hm	14. mar. 2009	rev 1.2
	removed double assignments

*)

END_FUNCTION_BLOCK

// POUs/Logic/gate logic/SHR1
FUNCTION SHR1 : DWORD
VAR_INPUT
	IN : DWORD;
	N : INT;
END_VAR
VAR CONSTANT
	temp : DWORD := 16#FFFF_FFFF;
END_VAR

(*
version 1.1	27 dec 2007
programmer 	hugo
tested by		tobias

SHR1 shifts N bits to the right filling the new bits with 1

*)

SHR1 := SHL(temp,32-N) OR SHR(IN,N);

(* revision history
hm	14.9.2007		rev 1.0
	original version

hm	27. dec 2007	rev 1.1
	changed code for better performance

*)

END_FUNCTION

// POUs/Mathematical/SIGMOID
FUNCTION SIGMOID : REAL
VAR_INPUT
	X : REAL;
END_VAR


(*
version 1.2	10. mar. 2009
programmer 	hugo
tested by		tobias

this function calculates the sigmoid function

*)

IF X > 20.0 THEN
	SIGMOID := 1.0;
ELSIF x < -85.0 THEN
	SIGMOID := 0.0;
ELSE
	SIGMOID := 1.0 / (1.0 + EXP(-X));
END_IF;


(* revision history
hm	10.12.2007		rev 1.0
	original version

hm	11. mar. 2008		rev 1.1
	extended range of valid inputs to +inv / -inv

hm 10. mar. 2009		rev 1.2
	real constants updated to new systax using dot																																																																																																																																																																																																																																																																																																																																																																																																																																																																																																																																																																																																																																																																																																																																																																																																																																																																																																																																																																																																																																																											

*)

END_FUNCTION

// POUs/Mathematical/SIGN_I
FUNCTION SIGN_I : BOOL
VAR_INPUT
	IN : DINT;
END_VAR


(*
version 1.3	27. oct. 2008
programmer 	hugo
tested by	tobias

this function return true if the integer input is negative

*)

SIGN_I := in.31;

(* revision history
hm 3.3.2007	rev 1.1
	changed method of function for better compatibility to other systems

hm	1.12.2007	rev 1.2
	changed code to improve performance

hm	27. oct. 2008	rev 1.3
	changed type of input to dint

*)

END_FUNCTION

// POUs/Engineering/automation/SIGNAL_4
FUNCTION_BLOCK SIGNAL_4
VAR_INPUT
	IN1 : BOOL;
	IN2 : BOOL;
	IN3 : BOOL;
	IN4 : BOOL;
	TS : TIME;
END_VAR
VAR_INPUT CONSTANT
	S1 : BYTE := 2#1111_1111;
	S2 : BYTE := 2#1111_0000;
	S3 : BYTE := 2#1010_1010;
	S4 : BYTE := 2#1010_0000;
END_VAR
VAR_OUTPUT
	Q : BOOL;
END_VAR
VAR
	sig : SIGNAL;
END_VAR

(*
version 1.0	13 dec 2007
programmer 	hugo
tested by		tobias

this function generates one out of 4 signals specified by bit patterns S1 .. S4.
the selected pattern will be shifted with the step time TS.
In1 has higher priority then In2 which has higher priority then IN3 and in4 has the lowest priority.
ts defaults to 128 ms if not specified.
*)

(* an alarm is present read system time first *)
(* check if an alarm is present if yes set sig to the alarm pattern otherwise exit the routine *)
IF in1 THEN
	sig(in := TRUE, sig := s1, TS := TS);
ELSIF in2 THEN
	sig(in := TRUE, sig := s2, TS := TS);
ELSIF in3 THEN
	sig(in := TRUE, sig := s3, TS := TS);
ELSIF in4 THEN
	sig(in := TRUE, sig := s4, TS := TS);
ELSE
	sig(in := FALSE);
END_IF;

(* set the output *)
Q := sig.Q;


(* revision history
hm	13.12.2007		rev 1.0
	original version

*)

END_FUNCTION_BLOCK

// POUs/Mathematical/SINC
FUNCTION SINC : REAL
VAR_INPUT
	X : REAL;
END_VAR


(*
version 1.2	10. mar. 2009
programmer 	hugo
tested by		tobias

this function calculates the sinc function.

*)

IF X = 0.0 THEN
	SINC := 1.0;
ELSE
	SINC := SIN(x) / x;
END_IF;


(* revision histroy
hm	11. mar. 2008	rev 1.0
	original version

hm	1.12.2007	rev 1.1
	changed code to improove performance

hm 10. mar. 2009	rev 1.2
	real constants updated to new systax using dot																																																																																																																																																																																																																																																																																																																																																																																																																																																																																																																																																																																																																																																																																																																																																																																																																																																																																																																																																																																																																																																											

*)

END_FUNCTION

// POUs/Mathematical/Geometry/SPHERE_V
FUNCTION SPHERE_V : REAL
VAR_INPUT
	rx : REAL;
END_VAR


(*
version 1.2	22. feb 2008
programmer 	hugo
tested by		tobias

sphere_V calculates the Volume of a Sphere


*)

sphere_V := 4.188790205 * Rx * RX * RX;

(* revision histroy
hm	16. oct 2007	rev 1.0
	original version

hm	4. dec 2007		rev 1.1
	changed code for better performance

hm	22. feb 2008		rev 1.2
	changed code for better performance
*)

END_FUNCTION

// POUs/Engineering/automation/SRAMP
FUNCTION_BLOCK SRAMP
VAR_INPUT
	X : REAL;
	A_UP : REAL;
	A_DN :REAL;
	VU_MAX : REAL;
	VD_MAX : REAL;
	LIMIT_HIGH : REAL;
	LIMIT_LOW : REAL;
	RST : BOOL;
END_VAR
VAR_OUTPUT
	Y : REAL;
	V : REAL;
END_VAR
VAR
	cycle_time : TC_S;
	init: BOOL;
END_VAR


(*
	version 1.1	11. mar. 2009
	programmer 	hugo
	tested by		tobias

RAMPS generates output signal which are slew rate and acceleration controlled.

*)

(* read the system_time in microseconds *)
cycle_time();

(* assure range of inputs *)
A_up := MAX(0.0, A_UP);
A_dn := MIN(0.0, A_dn);
VU_max := MAX(0.0, VU_max);
VD_max := MIN(0.0, VD_MAX);

(* calculate the output offset *)
IF rst OR NOT init THEN
	init := TRUE;
	Y := 0.0;
	V := 0.0;
ELSIF X = Y THEN
	v := 0.0;
ELSIF X > Y THEN
	(* output is too low >> ramp up and brake at the end *)
	(* accelerate the speed and limit to vu_max *)
	v := MIN(v + A_UP * cycle_time.TC, vu_max);
	(* calculate the max speed to be able to brake and select the lowest *)
	v := MIN(SQRT((Y-X) * 2.0 * A_DN), v);
	(* calculate the output and obey limits *)
	y := LIMIT(limit_low, y + MIN(v * cycle_time.TC, X-Y), limit_high);
ELSIF X < Y THEN
	(* output is too high >> ramp dn and brake at the end *)
	(* accelerate the speed and limit to vd_max *)
	v := MAX(v + A_DN * cycle_time.TC, vd_max);
	(* calculate the max speed to be able to brake and select the lowest *)
	v := MAX(-SQRT((Y-X) * 2.0 * A_UP), v);
	(* calculate the output and obey limits *)
	y := LIMIT(limit_low, y + MAX(v * cycle_time.TC, X-Y), limit_high);
END_IF;


(* revision history
hm	13. mar. 2008	rev 1.0
	original version

hm	11. mar. 2009	rev 1.1
	real constants updated to new systax using dot																																																																																																																																																																																																																																																																																																																																																																																																																																																																																																																																																																																																																																																																																																																																																																																																																																																																																																																																																																																																																																																											

*)

END_FUNCTION_BLOCK

// POUs/Engineering/measurements/TC_S
FUNCTION_BLOCK TC_S

VAR_OUTPUT
	TC : REAL;
END_VAR
VAR
	init: BOOL;
	tx: DWORD;
	last: DWORD;
END_VAR

(*
	version 1.2	11. mar. 2009
	programmer 	hugo
	tested by		tobias

TC_S delivers the time it was last called on the output TC in seconds.

*)

(* read system timer *)
tx := T_PLC_US();

IF NOT init THEN
	init := TRUE;
	TC := 0.0;
ELSE
	tc := DWORD_TO_REAL(tx - last)*1.0E-6;
END_IF;
last := tx;

(* revision history
hm	13. mar. 2008	rev 1.0
	original version

hm	16. mar 2008	rev 1.1
	added type conversion to avoid warnings under codesys 3.0

hm	11. mar. 2009	rev 1.2
	changed real constants to use dot syntax

*)

END_FUNCTION_BLOCK

// POUs/Logic/memory/STACK_16
FUNCTION_BLOCK STACK_16
VAR_INPUT
	Din : DWORD;
	E : BOOL := TRUE;
	RD : BOOL;
	WD : BOOL;
	RST : BOOL;
END_VAR
VAR_OUTPUT
	Dout : DWORD;
	EMPTY : BOOL := TRUE;
	FULL : BOOL;
END_VAR
VAR
	stack : ARRAY[0..n] OF DWORD;
	pt : INT;
END_VAR
VAR CONSTANT
	n : INT := 15;	(* changing this value will chage the number of stored elements in the fifo *)
END_VAR


(*
version 2.0	25. jul 2009
programmer 	hugo
tested by		oscat

16 Dword STACK memory

*)

IF RST THEN
	(* asynchronous reset for the fifo *)
	pt := 0;
	EMPTY := TRUE;
	FULL := FALSE;
	Dout := 0;
ELSIF E THEN
	IF NOT EMPTY AND RD THEN
		(* read one element *)
		pt := pt - 1;
		Dout := stack[pt];
		EMPTY := pt = 0;
		FULL := FALSE;
	END_IF;
	IF NOT FULL AND WD THEN
		(* write one element *)
		stack[pt] := Din;
		pt := pt + 1;
		FULL := pt > n;
		EMPTY := FALSE;
	END_IF;
END_IF;


(* revision history
hm	4. aug. 2006	rev 1.0
	original version

hm	19. feb 2008	rev 1.1
	performance improvements

hm	17. oct. 2008	rev 1.2
	deleted unnecessary init with 0

hm	27. oct. 2008	rev 1.3
	optimized performance

hm	25. jul 2009	rev 2.0
	changed inputs to allow simultsaneous read and write
*)

END_FUNCTION_BLOCK

// POUs/Logic/memory/STACK_32
FUNCTION_BLOCK STACK_32
VAR_INPUT
	Din : DWORD;
	E : BOOL := TRUE;
	RD : BOOL;
	WD : BOOL;
	RST : BOOL;
END_VAR
VAR_OUTPUT
	Dout : DWORD;
	EMPTY : BOOL := TRUE;
	FULL : BOOL;
END_VAR
VAR
	stack : ARRAY[0..n] OF DWORD;
	pt : INT;
END_VAR
VAR CONSTANT
	n : INT := 31;	(* changing this value will chage the number of stored elements in the fifo *)
END_VAR


(*
version 2.0	25. jul 2009
programmer 	hugo
tested by		oscat

32 Dword STACK memory
*)

IF RST THEN
	(* asynchronous reset for the fifo *)
	pt := 0;
	EMPTY := TRUE;
	FULL := FALSE;
	Dout := 0;
ELSIF E THEN
	IF NOT EMPTY AND RD THEN
		(* read one element *)
		pt := pt - 1;
		Dout := stack[pt];
		EMPTY := pt = 0;
		FULL := FALSE;
	END_IF;
	IF NOT FULL AND WD THEN
		(* write one element *)
		stack[pt] := Din;
		pt := pt + 1;
		FULL := pt > n;
		EMPTY := FALSE;
	END_IF;
END_IF;


(* revision history
hm	4. aug. 2006	rev 1.0
	original version

hm	19. feb 2008	rev 1.1
	performance improvements

hm	17. oct. 2008	rev 1.2
	deleted unnecessary init with 0

ks	27. oct. 2008	rev 1.3
	optimized performance

hm	25. jul 2009	rev 2.0
	changed inputs to allow simultsaneous read and write

*)

END_FUNCTION_BLOCK

// POUs/Engineering/signal processing/STAIR
FUNCTION STAIR : REAL
VAR_INPUT
	X : REAL;
	D : REAL;
END_VAR


(*
version 1.4	10. mar. 2009
programmer 	oscat
tested by		tobias

the function stair converts an anlog input signal to a staircase like output.
D is the step width for the output signal.
if D = 0 then the output follows the input without a chage.
*)

IF D > 0.0 THEN
	STAIR := DINT_TO_REAL(REAL_TO_DINT(X / D)) * D;
ELSE
	STAIR := X;
END_IF;



(* revision history
hm	28 jan 2007		rev 1.0
	original version

hm	27 dec 2007		rev 1.1
	changed code for better performance

hm	6. jan 2008		rev 1.2
	further performance improvement

hm	26. oct. 2008		rev 1.3
	optimized code

hm	10. mar. 2009	rev 1.4
	real constants updated to new systax using dot

*)

END_FUNCTION

// POUs/Engineering/signal processing/STAIR2
FUNCTION_BLOCK STAIR2
VAR_INPUT
	X : REAL;
	D : REAL;
END_VAR
VAR_OUTPUT
	Y: REAL;
END_VAR


(*
version 1.4	10. mar. 2009
programmer 	hugo
tested by		oscat

the function stair2 converts an anlog input signal to a staircase like output.
D is the step width for the output signal. the output will use D as a hysteresis for a stairchange.
if D = 0 then the output follows the input without a chage.
*)

IF D > 0.0 THEN
	IF X >= Y + D OR X <= Y - D THEN Y := FLOOR(X/D) * D; END_IF;
ELSE
	Y := X;
END_IF;



(* revision history
hm	28 jan 2007		rev 1.0
	original version

hm	27. dec 2007	rev 1.1
	changed code for better performance

hm	30. jun. 2008	rev 1.2
	added type conversions to avoid warnings under codesys 3.0																																																																																																																																																																																																																																																											

ks	26. oct. 2008	rev 1.3
	improved code

hm	10. mar. 2009	rev 1.4
	real constants updated to new systax using dot

*)

END_FUNCTION_BLOCK

// POUs/Logic/FF pulse triggered/STORE_8
FUNCTION_BLOCK STORE_8
VAR_INPUT
	Set : BOOL;
	D0,D1, D2, D3, D4, D5, D6, D7 : BOOL;
	Clr : BOOL;
	Rst : BOOL;
END_VAR
VAR_OUTPUT
	Q0, Q1, Q2, Q3, Q4, Q5, Q6, Q7 : BOOL;
END_VAR
VAR
	edge: BOOL;
END_VAR

(*
version 1.2	14. mar. 2009
programmer 	hugo
tested by		oscat

Store_4 stores up to 4 boolean inputs until a reset is clearing the outputs.
the respective output is set with a true at the respective input and stays true until a reset is generated.
a set input is used to set all outputs true at the same time, independent of their inputs.
a clear input is used to reset only the lowest priority of the outputs one at a time.
the lowest priority is q3.

*)

IF rst OR set THEN
	q0 := NOT rst;
	q1 := q0;
	q2 := q0;
	q3 := q0;
	q4 := q0;
	q5 := q0;
	q6 := q0;
	q7 := q0;
ELSE
	IF D0 THEN Q0 := TRUE; END_IF;
	IF D1 THEN Q1 := TRUE; END_IF;
	IF D2 THEN Q2 := TRUE; END_IF;
	IF D3 THEN Q3 := TRUE; END_IF;
	IF D4 THEN Q4 := TRUE; END_IF;
	IF D5 THEN Q5 := TRUE; END_IF;
	IF D6 THEN Q6 := TRUE; END_IF;
	IF D7 THEN Q7 := TRUE; END_IF;

	IF clr AND NOT edge THEN
		IF q0 THEN q0 := FALSE;
		ELSIF q1 THEN q1 := FALSE;
		ELSIF q2 THEN q2 := FALSE;
		ELSIF q3 THEN q3 := FALSE;
		ELSIF q4 THEN q4 := FALSE;
		ELSIF q5 THEN q5 := FALSE;
		ELSIF q6 THEN q6 := FALSE;
		ELSE q7 := FALSE;
		END_IF;
	END_IF;
	edge := clr;
END_IF;


(* revision history
hm	25.12.2007	rev 1.0
	original version

hm	30. oct. 2008	rev 1.1
	optimized performance

hm	14. mar. 2009	rev 1.2
	removed double assignments

*)

END_FUNCTION_BLOCK

// POUs/Logic/gate logic/SWAP_BYTE
FUNCTION SWAP_BYTE : WORD
VAR_INPUT
	IN : WORD;
END_VAR


(*
version 1.0	4 feb 2008
programmer 	hugo
tested by		tobias

This function swaps the high and low byte of the word in.

*)

SWAP_BYTE := ROL(in,8);


(* revision history
hm		4. feb 2008	rev 1.0
	original version

*)

END_FUNCTION

// POUs/Logic/gate logic/SWAP_BYTE2
FUNCTION SWAP_BYTE2 : DWORD
VAR_INPUT
	IN : DWORD;
END_VAR


(*
version 1.0	4 feb 2008
programmer 	hugo
tested by		tobias

This function reverses the byte order in the dword.

*)

Swap_Byte2 := (ROR(in,8) AND 16#FF00FF00) OR (ROL(in,8) AND 16#00FF00FF);

(* revision history
hm		4. feb 2008	rev 1.0
	original version

*)

END_FUNCTION

// POUs/Building/electrical/SWITCH_I
FUNCTION_BLOCK SWITCH_I
VAR_INPUT
	set : BOOL;
	in : BOOL;
	rst : BOOL;
END_VAR
VAR_INPUT CONSTANT
	T_debounce : TIME := T#10ms;
	T_reconfig : TIME := T#1s;
	T_on_max : TIME := T#0h;
END_VAR
VAR_OUTPUT
	Q : BOOL;
END_VAR
VAR
	state : BYTE;
	edge : BOOL;
	r_edge : BOOL;
	T_on : TIME;
	tx: TIME;
END_VAR

(*
version 1.1	15 sep 2007
programmer 	oscat
tested by	oscat

this is an intelligent switch interface which has an autodetect feature for in and it will detect the type of switch connected automatically
the input can be connected to low active pulses, high active pulses and on/off switch.
it will automatically adjust to the correct type without manual adjustment
a configurable debounce timer will debounce input signals
if t_on_max is set to anything other then 0 the output will be turned off after the max on time is reached.

*)

(* read system time *)
tx := DWORD_TO_TIME(T_PLC_MS());

(* asynchronous set and reset first *)
IF set AND NOT rst THEN
	Q := TRUE;
	T_on := tx;
ELSIF rst THEN
	Q := FALSE;
(* check FOR input edge AND start debounce timer *)
ELSIF (in XOR edge) AND NOT (state = 1) THEN
	state := 1;
	T_on := Tx;
(* edge was detected and debounce time elapsed *)
ELSIF (state = 1) AND (Tx - t_debounce >= T_on) THEN
	state := 2;
	(* react on rising or falling edge depending on r_edge *)
	IF r_edge XOR in THEN Q := NOT Q; END_IF;
(* wait for T_reconfig and adjust r_edge *)
ELSIF state = 2 AND Tx - t_reconfig >= T_on THEN
	r_edge := in;
END_IF;
IF Q AND T_on_max > t#0ms AND Tx >= T_on + T_on_max THEN
	Q := FALSE;
END_IF;
edge := in;

(* revision history

hm	4 aug 2006	rev 1.0
	original version

hm	15.9.2007	rev 1.1
	replaced Time() with T_PLC_MS for compatibility and performance reasons

*)

END_FUNCTION_BLOCK

// POUs/Building/electrical/SWITCH_X
FUNCTION_BLOCK SWITCH_X
VAR_INPUT
	IN1 : BOOL;
	IN2 : BOOL;
	IN3 : BOOL;
	IN4 : BOOL;
	IN5 : BOOL;
	IN6 : BOOL;
END_VAR
VAR_OUTPUT
	Q1 : BOOL;
	Q2 : BOOL;
	Q3 : BOOL;
	Q4 : BOOL;
	Q5 : BOOL;
	Q6 : BOOL;
	Q31 : BOOL;
	Q41 : BOOL;
	Q51 : BOOL;
	Q61 : BOOL;
	Q32 : BOOL;
	Q42 : BOOL;
	Q52 : BOOL;
	Q62 : BOOL;
END_VAR
VAR_INPUT CONSTANT
	t_debounce : TIME := t#50ms;
END_VAR
VAR
	init : BOOL;
	T1, T2, T3, T4, T5, T6 : TOF;
	tx: TIME;
	x1: BOOL;
	x2: BOOL;
	E1, E2 : BOOL;
END_VAR

(*
version 1.0	15 Feb 2007
programmer 	oscat
tested by	oscat

*)

(* initialize on startup *)
IF NOT init THEN
	init := TRUE;
	IF t_debounce < t#50ms THEN tx := t#50ms; ELSE tx := t_debounce; END_IF;
	T1(PT := Tx);
	T2(PT := Tx);
	T3(PT := Tx);
	T4(PT := Tx);
	T5(PT := Tx);
	T6(PT := Tx);
ELSE
	Q1 := FALSE;
	Q2 := FALSE;
	Q3 := FALSE;
	Q4 := FALSE;
	Q5 := FALSE;
	Q6 := FALSE;
	Q31 := FALSE;
	Q41 := FALSE;
	Q51 := FALSE;
	Q61 := FALSE;
	Q32 := FALSE;
	Q42 := FALSE;
	Q52 := FALSE;
	Q62 := FALSE;
END_IF;

(* read inputs and debounce *)
	T1(IN := IN1);
	T2(IN := IN2);
	T3(IN := IN3);
	T4(IN := IN4);
	T5(IN := IN5);
	T6(IN := IN6);

(* detect edge of IN1 and IN2 *)
IF t1.Q AND NOT E1 THEN X1 := TRUE; END_IF;
IF t2.Q AND NOT E2 THEN X2 := TRUE; END_IF;

IF t1.Q THEN
	IF t3.q THEN
		q31 := TRUE;
		X1 := FALSE;
	ELSIF t4.q THEN
		q41 := TRUE;
		X1 := FALSE;
	ELSIF t5.q THEN
		q51 := TRUE;
		X1 := FALSE;
	ELSIF t6.q THEN
		q61 := TRUE;
		X1 := FALSE;
	END_IF;
ELSIF t2.Q THEN
	IF t3.q THEN
		q32 := TRUE;
		X2 := FALSE;
	ELSIF t4.q THEN
		q42 := TRUE;
		X2 := FALSE;
	ELSIF t5.q THEN
		q52 := TRUE;
		X2 := FALSE;
	ELSIF t6.q THEN
		q62 := TRUE;
		X2 := FALSE;
	END_IF;
(* in1 was active alone *)
ELSIF NOT T1.Q AND E1 AND X1 THEN
	Q1 := TRUE;
	X1 := FALSE;
ELSIF NOT T2.Q AND E2 AND X2 THEN
	Q2 := TRUE;
	X2 := FALSE;
ELSIF T3.Q THEN
	Q3 := TRUE;
ELSIF T4.Q THEN
	Q4 := TRUE;
ELSIF T5.Q THEN
	Q5 := TRUE;
ELSIF T6.Q THEN
	Q6 := TRUE;
END_IF;

(* save state of in1 and in2 *)
E1 := T1.Q;
E2 := T2.Q;

END_FUNCTION_BLOCK

// POUs/Building/HLK/T_AVG24
FUNCTION_BLOCK T_AVG24
VAR_INPUT
	TS : INT;
	DTI : DT;
	RST : BOOL;
END_VAR
VAR_INPUT CONSTANT
	T_FILTER : TIME := T#10m;
	SCALE : REAL := 1.0;
	OFS : REAL;
END_VAR
VAR_OUTPUT
	TA : REAL;
	TP : BOOL;
END_VAR
VAR_IN_OUT
	T24 : REAL;
	T24_MAX : REAL;
	T24_MIN : REAL;
END_VAR
VAR
	samples : ARRAY[0..47] OF INT;
	pos : INT;
	init: BOOL;
	ft1 : FILTER_I;
	sum : DINT;
	last: DT;
END_VAR
VAR
	tmp_max : INT;
	tmp_min : INT;
	i: INT;
END_VAR

(*
version 1.2	13. mar. 2009
programmer 	hugo
tested by		oscat

this function calculates the averaged daytime temperature by taking 48 samples over one day.
a trigger tp will be true for one cycle when the output is updated.
using the input scale the outputs can be adjusted to different scales.

*)

(* first filter the sensor readings *)
ft1(X := TS, T := T_FILTER);

IF rst OR NOT init THEN
	init := TRUE;
	IF T24 = -1000.0 THEN t24 := INT_TO_REAL(ft1.Y) * 0.1; END_IF;
	FOR pos := 0 TO 47 DO
		samples[pos] := REAL_TO_INT(T24 * 10.0);
	END_FOR;
	pos := 0;
	sum := INT_TO_DINT(samples[0]) * 48;
	(* calculate the output value *)
	TA := (INT_TO_REAL(ft1.Y) * 0.1 + OFS) * SCALE;
	T24 := (DINT_TO_REAL(sum) * 0.00208333333333 + OFS) * SCALE;
	tp := TRUE;
ELSIF DT_TO_DWORD(dti) / 60 MOD 30 = 0 AND DTI > last THEN
	(* make sure we onlyexecute once every 30 mins *)
	last := DTI + T#1m;
	(* sample the temperature every 30 mins and store in ring buffer samples *)
	(* sum always holds the sum of the array *)
	(* subtract the oldest sample from sum *)
	sum := sum - INT_TO_DINT(samples[pos]);
	(* strore the new sample *)
	samples[pos] := ft1.Y;
	(* add the new sample to sum *)
	sum := sum + INT_TO_DINT(samples[pos]);
	(* increment the counter for the next sample *)
	pos := INC1(pos, 48);
	(* calculate the output value *)
	TA := (INT_TO_REAL(ft1.Y) * 0.1 + OFS) * SCALE;
	T24 := (DINT_TO_REAL(sum) * 0.00208333333333 + OFS) * SCALE;
	(* calculate the min and max over the last 24 hours *)
	tmp_max := -32000;
	tmp_min := 32000;
	FOR i := 0 TO 47 DO
		tmp_max := MAX(tmp_max, samples[i]);
		tmp_min := MIN(tmp_min, samples[i]);
	END_FOR;
	T24_MAX := (INT_TO_REAL(tmp_max) * 0.1 + OFS) * SCALE;
	T24_MIN := (INT_TO_REAL(tmp_min) * 0.1 + OFS) * SCALE;
	tp := TRUE;
ELSE
	tp := FALSE;
END_IF;





(* revision history
hm	3. nov. 2008	rev 1.0
	original version

hm	8. feb. 2009	rev 1.1
	changes sign of OFS
	added outputs t24_min and t24_max

hm	13. mar. 2009	rev 1.2
	improved code
*)

END_FUNCTION_BLOCK

// POUs/Mathematical/TANC
FUNCTION TANC : REAL
VAR_INPUT
	X : REAL;
END_VAR


(*
version 1.1	10. mar. 2009
programmer 	hugo
tested by		oscat

this function calculates the tanc function.

*)

IF X = 0.0 THEN
	TANC := 1.0;
ELSE
	TANC := TAN(x) / x;
END_IF;


(* revision histroy
hm	23. oct. 2008	rev 1.0
	original version

hm 10. mar. 2009	rev 1.1
	real constants updated to new systax using dot																																																																																																																																																																																																																																																																																																																																																																																																																																																																																																																																																																																																																																																																																																																																																																																																																																																																																																																																																																																																																																																											

*)

END_FUNCTION

// POUs/Mathematical/TANH
FUNCTION TANH : REAL
VAR_INPUT
	X : REAL;
END_VAR


(*
version 1.3	10. mar. 2009
programmer 	hugo
tested by		tobias

this function calculates the tangens hyperbolicus

*)

IF X > 20.0 THEN
	TANH := 1.0;
ELSIF X < -20.0 THEN
	TANH := -1.0;
ELSE
	TANH := 1.0 - 2.0 / (EXP(2.0 * x) + 1.0);
END_IF;


(* revision hisdtory
hm		12.1.2007		rev 1.0
	original version

hm		1.12.2007		rev 1.1
	changed code to improve performance

hm		10. mar 2008	rev 1.2
	corrected an error in formula
	extended range of valid inputs to +/- INV

hm 10. mar. 2009	rev 1.3
	real constants updated to new systax using dot																																																																																																																																																																																																																																																																																																																																																																																																																																																																																																																																																																																																																																																																																																																																																																																																																																																																																																																																																																																																																																																											

*)

END_FUNCTION

// POUs/Engineering/automation/TANK_LEVEL
FUNCTION_BLOCK TANK_LEVEL
VAR_INPUT
	LEVEL : BOOL;
	LEAK : BOOL;
	ACLR : BOOL;
END_VAR
VAR_INPUT CONSTANT
	MAX_VALVE_TIME : TIME;
	LEVEL_DELAY_TIME : TIME;
END_VAR
VAR_OUTPUT
	VALVE : BOOL;
	ALARM : BOOL;
	STATUS : BYTE;
END_VAR
VAR
	cx : ACTUATOR_COIL;
	tn : TON;
	tl : TONOF;
	open: BOOL;
END_VAR


(*
version 1.1	24 jul 2009
programmer 	hugo
tested by		tobias

*)

(* preprocess the level information *)
tl(in := level, T_ON := level_delay_time, T_OFF := level_delay_time);
open := tl.Q;

(* start logic *)
IF ALARM THEN
	(* check for ACLR if ALARM is present *)
	IF ACLR THEN
		ALARM := FALSE;
		STATUS := 101; (* aclr pressed *)
		cx(in := FALSE);
	END_IF;
	RETURN;
ELSIF LEAK THEN
	(* leakeage detected *)
	cx(in := FALSE);
	ALARM := TRUE;
	STATUS := 1;	(* leakeage error *)
ELSIF open THEN
	(* valve needs to be opened because level is too low *)
	cx(in := TRUE);
	STATUS := 102; (* valve open by low level *)
ELSE
	(* valve needs to be closed *)
	cx(in := FALSE);
	STATUS := 100; (* valve idle *)
END_IF;

(* check if valve is open too long and generate alarm if necessary *)
tn(in := cx.out AND (MAX_VALVE_TIME > T#0s), PT := MAX_VALVE_TIME);
IF tn.Q THEN
	ALARM := TRUE;
	STATUS := 2; (* overtime error *)
	cx(in := FALSE);
END_IF;

(* set output signal *)
VALVE := cx.out;


(* revision history
hm 27. feb 2007	rev 1.0
	original version

hm	24. jul 2009	rev 1.1
	changed parameters of tonof

*)

END_FUNCTION_BLOCK

// POUs/Logic/generators/TONOF
FUNCTION_BLOCK TONOF
VAR_INPUT
	IN : BOOL;
	  T_ON,T_OFF : TIME;
END_VAR
VAR_OUTPUT
	Q : BOOL;
END_VAR
VAR
   X : TON;
   old: BOOL;
   mode: BOOL;
END_VAR

(*
version 1.2	21. jul 2009
programmer 	hugo
tested by		tobias

TONOF generated a TON and TOF Delay for the Input N TON (T1) and TOF (T2) can be configured separately
*)

IF IN XOR old THEN
  X(IN := FALSE, PT := SEL(IN,T_OFF,T_ON));
  mode := IN;
  old := IN;
END_IF;
X(IN := TRUE);
IF X.Q THEN Q := mode;END_IF;

(* revision history
hm	10. dec 2007	rev 1.0
	original version

hm	17. sep. 2007	rev 1.1
	improved performance

hm	21. jul. 2009	rev 1.2
	fixed a timing probelm


*)

END_FUNCTION_BLOCK

// POUs/Building/HLK/TANK_VOL1
FUNCTION TANK_VOL1 : REAL
VAR_INPUT
	TR : REAL;
	TL : REAL;
	H : REAL;
END_VAR


(*
version 1.0	10. Mar 2010
programmer 	hugo
tested by		tobias

TANK_VOL1 calculates the volume of a tubular tank filled to level H.


*)

TANK_VOL1 := CIRCLE_SEG(TR, H) * TL;


(* revision histroy
hm	10. mar 2010	rev 1.0
	original version

*)

END_FUNCTION

// POUs/Building/HLK/TANK_VOL2
FUNCTION TANK_VOL2 : REAL
VAR_INPUT
	TR : REAL;
	H : REAL;
END_VAR


(*
version 1.0	10. Mar 2010
programmer 	hugo
tested by		tobias

TANK_VOL2 calculates the volume of a spherical tank filled to level H.

*)

TANK_VOL2 := math.PI * H * H * (TR - H/3.0);

(* revision histroy
hm	10. mar 2010	rev 1.0
	original version

*)

END_FUNCTION

// POUs/Engineering/measurements/TC_MS
FUNCTION_BLOCK TC_MS

VAR_OUTPUT
	TC : DWORD;
END_VAR
VAR
	init: BOOL;
	tx: DWORD;
	last: DWORD;
END_VAR

(*
	version 1.0	13 mar 2008
	programmer 	hugo
	tested by		tobias

TC_MS delivers the time it was last called on the output TC in Milliseconds.

*)

(* read system timer *)
tx := T_PLC_MS();

IF NOT init THEN
	init := TRUE;
	TC := 0;
ELSE
	tc := tx - last;
END_IF;
last := tx;

(* revision history
hm		13. mar. 2008	rev 1.0
	original version

*)

END_FUNCTION_BLOCK

// POUs/Engineering/measurements/TC_US
FUNCTION_BLOCK TC_US

VAR_OUTPUT
	TC : DWORD;
END_VAR
VAR
	init: BOOL;
	tx: DWORD;
	last: DWORD;
END_VAR

(*
	version 1.0	13 mar 2008
	programmer 	hugo
	tested by		tobias

TC_US delivers the time it was last called on the output TC in Microseconds.

*)

(* read system timer *)
tx := T_PLC_US();

IF NOT init THEN
	init := TRUE;
	TC := 0;
ELSE
	tc := tx - last;
END_IF;
last := tx;

(* revision history
hm		13. mar. 2008	rev 1.0
	original version

*)

END_FUNCTION_BLOCK

// POUs/Building/HLK/TEMP_EXT
FUNCTION_BLOCK TEMP_EXT
VAR_INPUT
	t_ext1 : REAL;
	t_ext2 : REAL;
	t_ext3 : REAL;
	t_ext_config : BYTE;
	dt_in : DT;
END_VAR
VAR_INPUT CONSTANT
	t_ext_min : REAL := -40.0;
	t_ext_max : REAL := 60.0;
	t_ext_default : REAL := -10.0;
	heat_period_start : DATE := D#1970-9-1;
	heat_period_stop : DATE := D#1970-4-30;
	cool_period_start : DATE := D#1970-4-1;
	cool_period_stop : DATE := D#1970-9-30;
	heat_start_temp_day : REAL := 15.0;
	heat_start_temp_night : REAL := 10.0;
	heat_stop_temp : REAL := 18.0;
	cool_start_temp_day : REAL := 26.0;
	cool_start_temp_night : REAL := 26.0;
	cool_stop_temp : REAL := 24.0;
	start_day : TOD := tod#09:00;
	start_night : TOD := tod#21:00;
	CYCLE_TIME : TIME := t#10m;
END_VAR
VAR_OUTPUT
	t_ext : REAL;
	heat : BOOL;
	cool : BOOL;
END_VAR
VAR
	tx: TIME;
	last_run: TIME;
	init: BOOL;
	cool_start: DATE;
	cool_stop: DATE;
	heat_start: DATE;
	heat_stop: DATE;
	xdate: DATE;
	day: BOOL;
END_VAR


(*
version 1.3	13. mar. 2009
programmer 	hugo
tested by		oscat

temp_ext measures and processes ext temperature and decides if heating or cooling is needed.

 the measurement of t_ext has 3 inputs which can be configured in different ways:
	t_ext_config = 0 means the ext temp is the avg of the 3 external temperatures, this mode is the default mode.
	t_ext_config = 1 means t_ext1 is used.
	t_ext_config = 2 means t_ext1 is used.
	t_ext_config = 3 means t_ext1 is used.
	t_ext_config = 4 means t_ext_default is used.
	t_ext_config = 5 means the lowest of the 3 external temperatures is used.
	t_ext_config = 6 means the higest externnal temperature is used.
	t_ext_config = 7 means the midlle external temperature is used, if there are only two working, the lowest is used.
	in any config mode, an external temperature higher then t_ext_max or lower then t_ext_min is ignored to prevent from temperatures caused by broken sensors or wires.
	if no external temperature is available, a default value (t_ext_default) is used.
	if you have only one external sensor, connect the 3 inputs to the same sensor, or select the right input with t_ext_config.

heating or cooling is enabled during heating / cooling period when the day or night start temperature is reached for at least the specified delay time and will be disabled after the stop temperature is reached. 
t_ext output can be used by other modules to determine the correct system temperature for heating or cooling.

*)

IF NOT init THEN
	init := TRUE;
	heat_start := SET_DATE(1972,MONTH_OF_DATE(heat_period_start),DAY_OF_MONTH(heat_period_start));
	heat_stop := SET_DATE(1972,MONTH_OF_DATE(heat_period_stop),DAY_OF_MONTH(heat_period_stop));
	cool_start := SET_DATE(1972,MONTH_OF_DATE(cool_period_start),DAY_OF_MONTH(cool_period_start));
	cool_stop := SET_DATE(1972,MONTH_OF_DATE(cool_period_stop),DAY_OF_MONTH(cool_period_stop));
END_IF;

(* read system time *)
tx := DWORD_TO_TIME(T_PLC_MS());

(* for efficiency exit isf this program has been executed less then 1min ago *)
IF tx - last_run < cycle_time THEN RETURN; END_IF;

(* calculate frequently used variables *)
xdate := SET_DATE(1972,MONTH_OF_DATE(DT_TO_DATE(dt_in)),DAY_OF_MONTH(DT_TO_DATE(dt_in)));
day := DT_TO_TOD(dt_in) >= start_day AND  DT_TO_TOD(dt_in) < start_night;

(* read the correct external temperature depending on the t_ext_config setting *)
t_ext := MULTI_IN(t_ext1, t_ext2, t_ext3, t_ext_default, t_ext_min, t_ext_max, t_ext_config);

(* dtermine heating *)
IF (heat_start <= heat_stop AND xdate >= heat_start AND xdate <= heat_stop) OR (heat_start > heat_stop AND (xdate >= heat_start OR xdate <= heat_stop)) THEN
	(* heating period id true check for temperature *)
	IF day AND t_ext <= heat_start_temp_day THEN
		heat := TRUE;
	ELSIF NOT day AND t_ext <= heat_start_temp_night THEN
		heat := TRUE;
	ELSIF t_ext >= heat_stop_temp THEN
		heat := FALSE;
	END_IF;
ELSE
	heat := FALSE;
END_IF;

(* dtermine cooling *)
IF (cool_start <= cool_stop AND xdate >= cool_start AND xdate <= cool_stop) OR (cool_start > cool_stop AND (xdate >= cool_start OR xdate <= cool_stop)) THEN
	(* cooling period is true check for temperature *)
	IF day AND t_ext >= cool_start_temp_day THEN
		cool := TRUE;
	ELSIF NOT day AND t_ext >= cool_start_temp_night THEN
		cool := TRUE;
	ELSIF t_ext <= cool_stop_temp THEN
		cool := FALSE;
	END_IF;
ELSE
	cool := FALSE;
END_IF;

last_run := tx;

(* revision history
hm	6 dec 2006	rev 1.0
	original version

hm	15.9.2007		rev 1.1
	replaced Time() with T_PLC_MS for compatibility and performance reasons

hm	7. oct. 2008	rev 1.2
	changed name of function month to month_of_date

hm	13. mar. 2009	rev 1.3
	real constants updated to new systax using dot

*)

END_FUNCTION_BLOCK

// POUs/Engineering/sensor/TEMP_NI
FUNCTION TEMP_NI : REAL
VAR_INPUT
	Res : REAL;
	R0 : REAL;
END_VAR


(*
version 1.5	10. mar. 2009
programmer 	hugo
tested by		tobias

this function returns the temperature for a nickel sensor in a range from -60..+180 °C *)

TEMP_NI := (SQRT(0.30085225 - 2.66E-3 * (R0 - Res)) - 0.5485) * 751.8796992;


(* revision history

hm 24.1.2007		rev 1.1
	deleted unused variable A, B, C

hm 10.9.2007		rev 1.2
	changed accuracy to 0.02 degrees to improove performace

hm 17. 12 2007	rev 1.3
	improovements for better performance and higher accuracy

hm	6. jan 2008	rev 1.4
	further performance improvement

hm	10. mar. 2009	rev 1.5
	removed nested comments

*)

END_FUNCTION

// POUs/Engineering/sensor/TEMP_NTC
FUNCTION TEMP_NTC : REAL
VAR_INPUT
	RES : REAL;
	RN : REAL;
	B : REAL;
END_VAR


(*
version 1.1	11. mar. 2009
programmer 	hugo
tested by		tobias

this function returs the temperature for a NTC sensor for a range from 0..85 °C.
RN is the resistance at 25 °C and B is a constant for the given sensor.

*)

IF res > 0.0 THEN
	TEMP_NTC := B * 298.15 / (B + LN(RES / RN) * 298.15) -273.15;
END_IF;


(* revision history

hm 30. dec. 2008	rev 1.0
	original version

hm	11. mar. 2009	rev 1.1
	changed real constants to use dot syntax

*)

END_FUNCTION

// POUs/Engineering/sensor/TEMP_PT
FUNCTION TEMP_PT : REAL
VAR_INPUT
	Res : REAL;
	R0 : REAL;
END_VAR
VAR CONSTANT
	A : REAL := 3.9083E-3 ;
	B : REAL := -5.775E-7;
	accuracy : REAL := 0.01;
END_VAR
VAR
	step: REAL := 50.0;
	X: REAL;
	Y: REAL;
	t1: REAL;
	pt : POINTER TO DWORD;
END_VAR

(*
version 1.7	11. mar. 2009
programmer 	hugo
tested by		oscat

this function returs the temperature for a platinum sensor for a range from -200..+850 °C *)

X := A * R0;
Y := B * R0;
IF Res >= R0 THEN
	t1 := X * X - 4.0 * Y * (R0 - Res);
	IF t1 < 0.0 THEN
		TEMP_PT := 10000.0;
	ELSE
		TEMP_PT := (-X + SQRT(t1)) / (2.0 * Y);
	END_IF;
ELSE
	pt := ADR(step);
	(* since the formula cannot be solved this is a successive approximation *)
	TEMP_PT := -100.0;
	WHILE step > accuracy DO
		(* test if result greater or less *)
		IF RES_PT(TEMP_PT, R0) < res THEN TEMP_PT := TEMP_PT + step; ELSE TEMP_PT := TEMP_PT - step; END_IF;
		pt^ := pt^ - 8388608;  (* this is a super fast divide by 2 method for non floating point CPUs *)
		(* the alternative code: step := step * 0.5; *)
	END_WHILE;
END_IF;

(* revision history

rev 1.1 hm 24.1.2007	
	deleted unused variable C

rev 1.2 hm 10.9.2007
	reduced accuracy to 0.02 to shorten execution time

rev 1.3	hm	2. dec 2007
	changed code for better performance

rev	1.4	hm	23. dec 2007
	avoid a negative square root if input values are wrong

rev 1.5 hm	5. jan 2008
	replaced / 2 with * 0.5 for better performance

hm	31. oct. 2008	rev 1.6
	improved performance

hm	11. mar. 2009	rev 1.7
	changed real constants to use dot syntax

*)

END_FUNCTION

// POUs/Engineering/sensor/TEMP_SI
FUNCTION TEMP_SI : REAL
VAR_INPUT
	Res : REAL;
	RS : REAL;
	TS : REAL;
END_VAR


(*
version 1.5	10. mar. 2009
programmer 	hugo
tested by		tobias

this function returs the temperature for a silicon sensor for a range from -60..+180 °C
for example KTY10 RS at TS normally 25 °C
*)

TEMP_SI := (-7.64E-3 + SQRT(Res / RS * 6.64E-5 - 0.803E-5)) * 30120.48193 + TS;



(* revision history

hm 24.1.2007		rev 1.1
	the function would only work for TS = 25, now it works for other values of ts.

hm 10.9.2007		rev 1.2
	changed the function to use successive approcimation to avoid an error generated by a sqrt from a negative result.
	changed accuracy to 0.02 degrees to shorten execution time

hm 17. 12 2007	rev 1.3
	improovements for better performance

hm	6. jan 2008	rev 1.4
	further performance improvement

hm	10. mar. 2009	rev 1.5
	removed nested comments

*)

END_FUNCTION

// POUs/String/TICKER
FUNCTION_BLOCK TICKER

VAR_INPUT
	N : INT;
	PT : TIME;
END_VAR

VAR_IN_OUT
	Text : STRING(STRING_LENGTH);
END_VAR

VAR_OUTPUT
	Display : STRING(STRING_LENGTH);
END_VAR
VAR
	delay : TP;
	step : INT;
END_VAR

(*
version 1.2	29. mar. 2008
programmer 	hugo
tested by		tobias

Ticker sends a substring of text with length N every TD Milliseconds to generate a ticker. 

*)


(* generate next ticker when delay is low *)
IF N < LEN(text) THEN
	IF NOT delay.Q THEN
		(* increase step for next tick *)
		step := step + 1;
		IF step > LEN(text) THEN step := 1; END_IF;
		(* extract dispay from text *)
		display := MID(text, N, step);
		(* set delay timer for next tick *)
		delay(in := TRUE, PT := PT);
	ELSE;
		(* execute delay timer *)
		delay(in := FALSE);
	END_IF;
ELSE
	display := text;
END_IF;
(* revision history
hm	4. dec. 2007	rev 1.0
	original version

hm	15. dec. 2007	rev 1.1
	step now starts at 1 instaed of 0

hm	29. mar. 2008	rev 1.2
	changed STRING to STRING(STRING_LENGTH)
*)

END_FUNCTION_BLOCK

// POUs/Building/electrical/TIMER_2
FUNCTION_BLOCK TIMER_2
VAR_INPUT
	DT_in : DT;
	start : TOD;
	duration : TIME;
	mode : BYTE;
	HOLIDAY : BOOL;
END_VAR
VAR_OUTPUT
	Q : BOOL;
END_VAR
VAR
	last_check : TIME;
	dat : DATE;
	daytime : TOD;
	activation: TIME;
	tx: TIME;
	enabled: BOOL;
	init: BOOL;
	wday : INT;
END_VAR

VAR RETAIN
	run_date : DATE;
END_VAR

(*
version 1.4	20. oct. 2008
programmer 	oscat
tested by	oscat

this timer generated programmabe output pulses per day, week, month and so on.
the mode input determines on which days the timer will be active.
	mode = 0			never
	mode = 1..7			monday .. sunday
	mode = 11			every day
	mode = 12			every second day
	mode = 13			every 3rd day
	mode = 14			every 4th day
	mode = 15			every 5th day
	mode = 16 			every 6th day
	mode = 20			only monday - friday
	mode = 21			only sat - sunday
	mode = 22			workdays only
	mode = 23			holidays and weekend
	mode = 24			holidays only
	mode = 25			every 1st day of the month
	mode = 26			every last day of the month
	mode = 27			every 31 of december
	mode = 28			every 1st of january

a holiday input can be used to supply holiday information to the module.
*)

(* read system time *)
tx := DWORD_TO_TIME(T_PLC_MS());

IF NOT init THEN
	init := TRUE;
	last_check := tx - t#100ms;
END_IF;

(* for performance resons exit if execution is not necessary *)
IF tx - last_check < T#100ms THEN RETURN; END_IF;

(* calculate temp variables *)
dat := DT_TO_DATE(dt_in);
daytime := DT_TO_TOD(dt_in);
wday := DAY_OF_WEEK(dat);

(* calculate if any action is necessary today *)
CASE mode OF
	1..7:	(* mondays to fridays *)
		enabled := wday = BYTE_TO_INT(mode);
	11:	(* every day *)
		enabled := TRUE;
	12..16:	(* every nth day *)
		enabled := (DATE_TO_DWORD(dat)/86400) MOD (mode - 10) = 0;
	20:	(* monday - friday *)
		enabled := wday <= 5;
	21:	(* saturday and sunday *)
		enabled := wday > 5;
	22: (* workdays only *)
		enabled := wday <= 5 AND NOT holiday;
	23:	(* holidays and weekends *)
		enabled := wday > 5 OR holiday;
	24:	(* holidays only *)
		enabled := holiday;
	25:	(* 1st day of the month *)
		enabled := DAY_OF_MONTH(dat) = 1;
	26:	(* last day of month *)
		enabled := DAY_OF_MONTH(dat + t#1d) = 1;
	27:	(* 31st of december *)
		enabled := DAY_OF_MONTH(dat) = 31 AND MONTH_OF_DATE(dat) = 12;
	28:	(* 1st of january *)
		enabled := DAY_OF_YEAR(dat) = 1;
ELSE
	enabled := FALSE;
END_CASE;

(* set output if necessary *)
IF enabled AND NOT Q AND daytime >= start AND run_date <> dat THEN
	Q := TRUE;
	activation := tx;
	run_date := dat;
ELSIF Q AND tx - activation >= duration THEN
	Q := FALSE;
END_IF;
last_check := Tx;


(* revision history
hm 22.2.2007		rev 1.1
	changed VAR RETAIN PERSISTENT to VAR RETAIN for better compatibility
	wago lon contollers do not support persisitent

hm	15.9.2007		rev 1.2
	replaced Time() with T_PLC_MS for compatibility and performance reasons

hm	7. oct. 2008	rev 1.3
	changed function month to month_of_date

hm	20. oct. 2008	rev 1.4
	improved performance
	deleted unnecessary trunc

hm	22. dec. 2008	rev 1.5
	make sure timer_2 is executed in the first cycle

*)

END_FUNCTION_BLOCK

// POUs/Building/electrical/TIMER_EVENT_DECODE
FUNCTION TIMER_EVENT_DECODE : TIMER_EVENT
VAR_INPUT
	EVENT : STRING(STRING_LENGTH);
	LANG :	INT;
END_VAR
VAR
	pos: INT;
	start : INT;
	stop: INT;
	pt : POINTER TO ARRAY[1..255] OF BYTE;
	step: INT;
	tmp : STRING(60);
END_VAR



(*
version 1.1	25. oct. 2008
programmer 	hugo
tested by	oscat

STRING_TO_TIMER_EVENT converts a string to a timer event structure.

*)

(* a timer event is specified as follows:
	$typ;ch;day;start;duration;land;lor#
$ 		= start of definition
typ 	= type of definition	(number)
channel	= channel number		(number)
day 	= day number			(number)
start	= start time			(time of day)
duration= duration of event		(time)
land	= mask for output AND	(8bit value)
lor		= mask for ourput OR	(8bit value)
#		= end of definition
*)

(* check for start and ending character *)
IF (LEFT(event,1) <> '<') AND (RIGHT(event,1) <> '>') THEN RETURN; END_IF;
stop := LEN(event);
pt := ADR(event);
start := 2;

(* parse the string for next ; *)
FOR pos := 2 TO stop DO
	IF pt^[pos] = 59 OR pt^[pos] = 62 THEN
		tmp := MID(event, pos - start, start);
		CASE step OF
			0:	(* read type *)
				TIMER_EVENT_DECODE.typ := FSTRING_TO_BYTE(tmp);

			1:	(* read channel *)
				TIMER_EVENT_DECODE.channel := FSTRING_TO_BYTE(tmp);

			2:	(* read day *)
				IF IS_CC(tmp,'0123456789abcdefABCDEF#') THEN
					TIMER_EVENT_DECODE.day := FSTRING_TO_BYTE(tmp);
				ELSIF TIMER_EVENT_DECODE.typ = 2 THEN
					TIMER_EVENT_DECODE.DAY := FSTRING_TO_WEEK(tmp, LANG);
				ELSE
					TIMER_EVENT_DECODE.DAY := INT_TO_BYTE(FSTRING_TO_WEEKDAY(tmp, LANG));
				END_IF;

			3:	(* read start *)
				TIMER_EVENT_DECODE.start := STRING_TO_TOD(tmp);

			4:	(* read duaration *)
				TIMER_EVENT_DECODE.duration := STRING_TO_TIME(tmp);

			5:	(* read land *)
				TIMER_EVENT_DECODE.land := FSTRING_TO_BYTE(tmp);

			6:	(* read lor *)
				TIMER_EVENT_DECODE.LOR := FSTRING_TO_BYTE(tmp);
		END_CASE;
		start := pos + 1;
		step := step + 1;
	END_IF;
END_FOR;




(* revision history
hm	17. jun 2008	rev 1.0
	original version

hm	25. oct. 2008	rev 1.1
	adding input lang for language selection
*)

END_FUNCTION

// POUs/Building/electrical/TIMER_EXT
FUNCTION_BLOCK TIMER_EXT
VAR_INPUT
	ENA : BOOL := TRUE;
	ON : BOOL;
	OFF : BOOL;
	MAN : BOOL;
	SWITCH : BOOL;
	DT_IN : DT;
	SUN_RISE : TOD;
	SUN_SET : TOD;
	HOLIDAY : BOOL;
END_VAR
VAR_INPUT CONSTANT
	T_DEBOUNCE : TIME := T#100ms;
	T_RISE_START : TIME;
	T_RISE_STOP : TIME;
	T_SET_START : TIME;
	T_SET_STOP : TIME;
	T_DAY_START : TOD;
	T_DAY_STOP : TOD;
	ENABLE_SATURDAY : BOOL;
	ENABLE_SUNDAY : BOOL;
	ENABLE_HOLIDAY : BOOL;
END_VAR
VAR_OUTPUT
	Q : BOOL;
	STATUS: BYTE;
END_VAR
VAR
	mx : MANUAL_2;
	deb : DEBOUNCE;
	tdx: TOD;
	wdx: INT;
	tc : TIME;
	tx: DWORD;
	tl: DWORD;
	qx: BOOL;
	init: BOOL;
END_VAR

(*
version 1.1	6. nov. 2008
programmer 	oscat
tested by	tobias

TIMER_EXT is a twilight timer.
the timer can be programmed to switch lights or other equippment or during twilight times.
in addition to the automatik mode the timer can be stopped and started by a switch at any given time.
An enable input ENA can be used for external control.
two inputs ON and OFF can be used to statically control the output.
the timer can be programmed to work on saturdays, sundays and holidays if required.

*)

(* lösche die millisekunden bei sunrise und sunset *)
SUN_RISE := DWORD_TO_TOD(TOD_TO_DWORD(SUN_RISE) / 1000 * 1000);
SUN_SET := DWORD_TO_TOD(TOD_TO_DWORD(SUN_SET) / 1000 * 1000);

(* measure cycle time tc and make sure this circuitry is not called more then once in 200ms*)
tx := T_PLC_MS();
IF NOT init THEN
	init := TRUE;
	tl := tx;
END_IF;
tc := DWORD_TO_TIME(tx - tl);
IF tc < t#200ms THEN RETURN; END_IF;
tl := tx;

(* debounce *)
deb(in := SWITCH, TD := T_DEBOUNCE, PM := TRUE);

(* read time of day and strip off all milliseconds *)
tdx := DT_TO_TOD(dt_in);
wdx := DAY_OF_WEEK(DT_TO_DATE(dt_in));

(* automatic output control *)
IF deb.Q THEN
	qx := NOT qx;
	status := 110;
ELSIF holiday AND NOT enable_holiday THEN
	qx := FALSE;
ELSIF wdx = 6 AND NOT enable_saturday THEN
	qx := FALSE;
ELSIF wdx = 7 AND NOT enable_sunday THEN
	qx := FALSE;
ELSIF T_day_start > TOD#00:00 AND tdx - T_DAY_START <= tc THEN
	(* turn on at specified daytime *)
	qx := TRUE;
	status := 111;
ELSIF T_DAY_STOP > TOD#00:00 AND tdx - T_DAY_STOP <= tc THEN
	(* turn off at specific daytime *)
	qx := FALSE;
	status := 112;
ELSIF T_RISE_START > T#0s AND tdx - SUN_RISE + T_RISE_START <= tc THEN
	(* turn on before sunrise *)
	qx := TRUE;
	status := 113;
ELSIF T_RISE_STOP > T#0s AND tdx - SUN_RISE - T_RISE_STOP <= tc THEN
	(* turn off after sunrise *)
	qx := FALSE;
	status := 114;
ELSIF T_SET_start > T#0s AND tdx - SUN_SET + T_SET_START <= tc THEN
	(* turn on before sunset *)
	qx := TRUE;
	status := 115;
ELSIF T_SET_STOP > t#0s AND tdx - SUN_SET - T_SET_STOP <= tc THEN
	(* turn off after sunset *)
	qx := FALSE;
	status := 116;
END_IF;


(* mnaual and output control *)
mx(in := qx, ena := ENA, on := ON, off := OFF, man := MAN);
Q := mx.Q;

(* set the status output *)
IF mx.STATUS > 100 THEN status := mx.STATUS; END_IF;



(*
hm 	7. oct. 2008	rev 1.0
	original version

hm	6. nov. 2008	rev 1.1
	added default = true for ena input
*)

END_FUNCTION_BLOCK

// POUs/Building/electrical/TIMER_P4
FUNCTION_BLOCK TIMER_P4
VAR_INPUT
	DTIME : DT;
	TREF_0 : TOD;
	TREF_1 : TOD;
	HOLY : BOOL;
	L0, L1, L2, L3 : BOOL;
	OFS : BYTE;
	ENQ : BOOL;
	MAN : BOOL;
	MI : BYTE;
	RST : BOOL;
END_VAR
VAR_IN_OUT
	PROG : ARRAY[0..array_max] OF TIMER_EVENT;
END_VAR
VAR_OUTPUT
	Q0, Q1, Q2, Q3 : BOOL;
	STATUS : BYTE;
END_VAR
VAR CONSTANT
	array_max : INT := 63;
	channel_max : INT := 3;
END_VAR
VAR
	day_start : DT;
	start : DT;
	event : TIMER_EVENT;
	pos : INT;
	last_execute: DT;
	current_day : DINT;
	mask: BYTE;
	ma : ARRAY[0..channel_max] OF BYTE;
	mo : ARRAY[0..channel_max] OF BYTE;
	qn : ARRAY[0..channel_max] OF BOOL;
	qs : ARRAY[0..channel_max] OF BOOL;
	channel: INT;
	tx: TOD;
END_VAR


(*
version 1.4	26. jan. 2011
programmer 	hugo
tested by	oscat

TIMER_P4 is a programmable universal timer.
*)

(* for performance reasons we only execute the code at the beginning of a new second *)

IF RST THEN
	(* reset all events to last active on 1.1.1970 *)
	last_execute := DT#1970-1-1-00:00;
	FOR pos := 0 TO ARRAY_MAX DO
		IF (PROG[pos].CHANNEL >= OFS) AND (PROG[pos].CHANNEL < (OFS + 4)) THEN PROG[pos].LAST := last_execute; END_IF;
	END_FOR;

	(* reset all set markers and logic masks *)
	FOR pos := 0 TO channel_max DO
		qs[pos] := FALSE;
	END_FOR;

(* normal operation *)
ELSIF dtime <> last_execute THEN
	(* save the actual second for next execution test *)
	last_execute := DTIME;

	(* calculate dt for the start of the day to be used in comparisons *)
	day_start := DATE_TO_DT(DT_TO_DATE(DTIME));

	(* set all qn to FALSE *)
	FOR pos := 0 TO channel_max DO qn[pos] := FALSE; END_FOR;

	(* search the array PROG for timer events *)
	FOR pos := 0 TO ARRAY_MAX DO
		event := prog[pos];
		channel := event.CHANNEL - OFS;
		IF (event.TYP > 0) AND (channel >= 0) AND (channel <= channel_max) THEN
			ma[channel] := event.LAND;
			mo[channel] := event.LOR;
			CASE event.TYP OF
				1:	(* daily event *)
					start := day_start + TOD_TO_TIME(event.start);
					qn[channel] := dtime >= start AND dtime <= start + event.DURATION;

				2: 	(* event by selected weekdays *)
					IF (SHR(BYTE#128, DAY_OF_WEEK(DT_TO_DATE(Dtime))) AND event.DAY) > 0 THEN
						start := day_start + TOD_TO_TIME(event.start);
						qn[channel] := dtime >= start AND dtime <= start + event.DURATION;
					END_IF;

				3:	(* event every N days *)
					IF current_day MOD event.DAY = 0 THEN
						start := day_start + TOD_TO_TIME(event.start);
						qn[channel] := dtime >= start AND dtime <= start + event.DURATION;
					END_IF;

				10:	(* weekly event exactly once a week the weekday is specified in day, 1= mo *)
					IF DAY_OF_WEEK(DT_TO_DATE(DTIME)) = BYTE_TO_INT(event.DAY) THEN
						start := day_start + TOD_TO_TIME(event.start);
						qn[channel] := dtime >= start AND dtime <= start + event.DURATION;
					END_IF;

				20:	(* monthly event *)
					IF DAY_OF_MONTH(DT_TO_DATE(DTIME)) = BYTE_TO_INT(event.DAY) THEN
						start := day_start + TOD_TO_TIME(event.start);
						qn[channel] := dtime >= start AND dtime <= start + event.DURATION;
					END_IF;

				21:	(* event on last day of month *)
					IF DT_TO_DATE(DTIME) = MONTH_END(DT_TO_DATE(dtime)) THEN
						start := day_start + TOD_TO_TIME(event.start);
						qn[channel] := dtime >= start AND dtime <= start + event.DURATION;
					END_IF;

				30:	(* yearly event on a specific day specified in day *)
					IF DAY_OF_YEAR(DT_TO_DATE(DTIME)) = BYTE_TO_INT(event.DAY) THEN
						start := day_start + TOD_TO_TIME(event.start);
						qn[channel] := dtime >= start AND dtime <= start + event.DURATION;
					END_IF;

				31:	(* event on last day of year *)
					IF DT_TO_DATE(DTIME) = YEAR_END(YEAR_OF_DATE(DT_TO_DATE(dtime))) THEN
						start := day_start + TOD_TO_TIME(event.start);
						qn[channel] := dtime >= start AND dtime <= start + event.DURATION;
					END_IF;

				40:	(* event on leap days *)
					IF LEAP_DAY(DT_TO_DATE(dtime)) THEN
						start := day_start + TOD_TO_TIME(event.start);
						qn[channel] := dtime >= start AND dtime <= start + event.DURATION;
					END_IF;

				41: (* event on holidays *)
					IF HOLY THEN
						start := day_start + TOD_TO_TIME(event.start);
						qn[channel] := dtime >= start AND dtime <= start + event.DURATION;
					END_IF;

				42: (* event on holidays and weekends *)
					IF (Holy OR (DAY_OF_WEEK(DT_TO_DATE(dtime)) = 6) OR (DAY_OF_WEEK(DT_TO_DATE(dtime)) = 7)) THEN
						start := day_start + TOD_TO_TIME(event.start);
						qn[channel] := dtime >= start AND dtime <= start + event.DURATION;
					END_IF;

				43:	(* event on workdays Mo-FR and no holiday *)
					IF DAY_OF_WEEK(DT_TO_DATE(dtime)) < 6 THEN
						start := day_start + TOD_TO_TIME(event.start);
						qn[channel] := dtime >= start AND dtime <= start + event.DURATION;
					END_IF;

				50: (* event after reference time *)
					CASE prog[pos].DAY OF
						0:	tx := tref_0;
						1:	tx := tref_1;
					ELSE
						tx := TOD#00:00;
					END_CASE;
					start := day_start + TOD_TO_TIME(tx) + TOD_TO_TIME(event.start);
					qn[channel] := dtime >= start AND dtime <= start + event.DURATION;

				51:	(* event before reference time *)
					CASE prog[pos].DAY OF
						0:	tx := tref_0;
						1:	tx := tref_1;
					ELSE
						tx := TOD#00:00;
					END_CASE;
					start := day_start + TOD_TO_TIME(tx) - TOD_TO_TIME(event.start);
					qn[channel] := dtime >= start AND dtime <= start + event.DURATION;

				52 : (* set output at specific time + offset  *)
					CASE prog[pos].DAY OF
						0:	tx := tref_0;
						1:	tx := tref_1;
					ELSE
						tx := TOD#00:00;
					END_CASE;
					start := day_start + TOD_TO_TIME(tx) + TOD_TO_TIME(event.start);
					IF dtime >= start AND day_start > event.LAST THEN
						qs[channel] := TRUE;
						prog[pos].LAST := day_start;
					END_IF;

				53 : (* reset output at specific time + offset *)
					CASE prog[pos].DAY OF
						0:	tx := tref_0;
						1:	tx := tref_1;
					ELSE
						tx := TOD#00:00;
					END_CASE;
					start := day_start + TOD_TO_TIME(tx) + TOD_TO_TIME(event.start);
					IF dtime >= start AND day_start > event.LAST THEN
						qs[channel] := FALSE;
						prog[pos].LAST := day_start;
					END_IF;

				54 : (* set output at specific time - offset  *)
					CASE prog[pos].DAY OF
						0:	tx := tref_0;
						1:	tx := tref_1;
					ELSE
						tx := TOD#00:00;
					END_CASE;
					start := day_start + TOD_TO_TIME(tx) - TOD_TO_TIME(event.start);
					IF dtime >= start AND day_start > event.LAST THEN
						qs[channel] := TRUE;
						prog[pos].LAST := day_start;
					END_IF;

				55 : (* reset output at specific time - offset *)
					CASE prog[pos].DAY OF
						0:	tx := tref_0;
						1:	tx := tref_1;
					ELSE
						tx := TOD#00:00;
					END_CASE;
					start := day_start + TOD_TO_TIME(tx) - TOD_TO_TIME(event.start);
					IF dtime >= start AND day_start > event.LAST THEN
						qs[channel] := FALSE;
						prog[pos].LAST := day_start;
					END_IF;
			END_CASE;
		END_IF;
	END_FOR;
END_IF;

(* prepare the logical input mask *)
mask := 255;
mask.0 := L0;
mask.1 := L1;
mask.2 := L2;
mask.3 := L3;

(* set the outputs *)
Q0 := ENQ AND ((qn[0] OR qs[0]) AND ((ma[0] AND mask) = ma[0]) OR ((mo[0] AND mask) > 0) OR (man AND MI.0));
Q1 := ENQ AND ((qn[1] OR qs[1]) AND ((ma[1] AND mask) = ma[1]) OR ((mo[1] AND mask) > 1) OR (man AND MI.1));
Q2 := ENQ AND ((qn[2] OR qs[2]) AND ((ma[2] AND mask) = ma[2]) OR ((mo[2] AND mask) > 2) OR (man AND MI.2));
Q3 := ENQ AND ((qn[3] OR qs[3]) AND ((ma[3] AND mask) = ma[3]) OR ((mo[3] AND mask) > 3) OR (man AND MI.3));

(* set status *)
IF NOT enq THEN
	status := 100;
ELSIF man THEN
	status := 101;
ELSE
	status := 102;
END_IF;



(* revision history
hm	17. jun 2008	rev 1.0
	original version

hm	9. oct. 2008	rev 1.1
	changed function year to year_of_date
	changed function weekday to day_of_week
	changed structure of program to be more efficient
	changed input DIS to ENQ

hm	18. oct. 2008	rev 1.2
	changed type of input OFS from int to byte
	added typecasts to avoid warnings

hm	28. feb. 2009	rev 1.3
	array was not correctly initialized

hm	26. jan 2011	rev 1.4
	changed code to allow events over midnight
*)

END_FUNCTION_BLOCK

// POUs/Time&Date/YEAR_END
FUNCTION YEAR_END : DATE
VAR_INPUT
	y : INT;
END_VAR


(*
version 1.1	24. jan. 2011
programmer 	hugo
tested by	oscat

returs the date of december 31st for the given year  
the function works for dates from 1970 - 2099 

*)

YEAR_END := DWORD_TO_DATE(SHR(INT_TO_DWORD(y) * 1461 - 2876712, 2) * 86400);



(* revision history
hm	15. jun. 2008	rev 1.0
	original version

hm	24. jan 2011	rev 1.1
	improved performance
*)

END_FUNCTION

// POUs/Logic/generators/TOF_1
FUNCTION_BLOCK TOF_1
VAR_INPUT
	IN : BOOL;
	PT : TIME;
	RST : BOOL;
END_VAR
VAR_OUTPUT
	Q : BOOL;
END_VAR
VAR
	tx : TIME;
	start : TIME;
END_VAR

(*
version 1.0	17. jul. 2008
programmer 	hugo
tested by	oscat

TOF_1 will extend a pulse on input in for PT seconds.
in addition the timer can be cleared asynchronously with rst.
TOF_1 is the same function as TOF from the standard LIB except the asynchronous reset input.

*)

(* read system timer *)
tx := DWORD_TO_TIME(T_PLC_MS());

IF RST THEN
	Q := FALSE;
ELSIF IN THEN
	Q := TRUE;
	start := tx;
ELSIF tx - start >= PT THEN
	Q := FALSE;
END_IF;




(* revision history
hm	17. jul. 2008	rev 1.0
	original version

*)

END_FUNCTION_BLOCK

// POUs/Mathematical/Geometry/TRIANGLE_A
FUNCTION TRIANGLE_A : REAL
VAR_INPUT
	S1 : REAL;
	A : REAL;
	S2 : REAL;
	S3 : REAL;
END_VAR


(*
version 1.2	10. mar. 2009
programmer 	hugo
tested by		tobias

triangle_A calculates the Area of a triangle.
if any input is 0 it will be neglected and the are will be calculated from eiter:
two sides and an angle (s1 and S2 and the angle A1) or 3 sides.


*)

IF A = 0.0 THEN
	TRIANGLE_A := SQRT((s1+s2+S3) * (s1+s2-S3) * (S2+S3-S1) * (S3+S1-S2)) * 0.25;
ELSE
	TRIANGLE_A := S1 * S2 * SIN(RAD(A)) * 0.5;
END_IF;

(* revision histroy
hm	16. oct 2007	rev 1.0
	original version

hm	22. feb 2008	rev 1.1
	improved performance

hm	10. mar. 2009	rev 1.2
	changed syntax of real constants to 0.0

*)

END_FUNCTION

// POUs/String/TRIM1
FUNCTION TRIM1 : STRING(STRING_LENGTH)
VAR_INPUT
	str : STRING(STRING_LENGTH);
END_VAR
VAR
	pos: INT;
END_VAR

(*
version 1.2	29. mar. 2008
programmer 	hugo
tested by		tobias

the function replaces all multiple blanks within a string by only one blank.
leading and ending blanks will be deleted

*)

TRIM1 := str;
REPEAT
	pos := FIND(trim1,'  ');
	IF pos > 0 THEN TRIM1 := REPLACE(TRIM1,' ',2,pos); END_IF;
UNTIL pos = 0	END_REPEAT;
(* beginning and ending blanks need to be stripped off *)
IF LEFT(trim1,1) = ' ' THEN trim1 := DELETE(trim1,1,1); END_IF;
IF RIGHT(trim1,1) = ' ' THEN trim1 := DELETE(trim1,1,LEN(trim1)); END_IF;


(* revision histroy
hm	4. feb. 2008    rev 1.0
	original release

hm	20. mar. 2008	rev 1.1
	avoid to call replace with pos = 0 because some systems will produce an error

hm	29. mar. 2008	rev 1.2
	changed STRING to STRING(STRING_LENGTH)
*)

END_FUNCTION

// POUs/String/TRIME
FUNCTION TRIME : STRING(string_length)
VAR_INPUT
	str : STRING(STRING_LENGTH);
END_VAR


(*
version 1.0	28. mar. 2008
programmer 	hugo
tested by	tobias

this function deletes all leading and ending blanks of a string.

*)

TRIME := str;
(* beginning blanks need to be stripped off *)
WHILE LEFT(TRIME,1) = ' ' DO
	TRIME := DELETE(TRIME,1,1);
END_WHILE;

(* ending blanks need to be stripped off *)
WHILE RIGHT(TRIME,1) = ' ' DO
	TRIME := DELETE(TRIME,1,LEN(TRIME));
END_WHILE;


(* revision histroy
hm	28. mar. 2008	rev 1.0
	original release

*)

END_FUNCTION

// POUs/Engineering/automation/TUNE
FUNCTION_BLOCK TUNE
VAR_INPUT
	SET : BOOL;
	SU, SD : BOOL;
	RST : BOOL;
END_VAR
VAR_INPUT CONSTANT
	SS : REAL := 0.1;
	Limit_L : REAL;
	LIMIT_H : REAL := 100.0;
	RST_val : REAL;
	SET_val : REAL := 100.0;
	T1 : TIME := T#500ms;
	T2 : TIME := T#2s;
	S1 : REAL := 2.0;
	S2 : REAL := 10.0;
END_VAR
VAR_OUTPUT
	Y : REAL;
END_VAR
VAR
	tx : DWORD;
	start, start2 : DWORD;
	state : INT;
	in : BOOL;
	step : REAL;
	SPEED : REAL;
	Y_start : REAL;
	Y_start2: REAL;
END_VAR

(*
version 1.2	11. mar. 2009
programmer 	hugo
tested by		tobias

tune generates an output signal which is set by input switches.
up to 4 switsches can be used to tune the signal up or down.

*)

(* read system time *)
tx := T_PLC_MS();

IF rst THEN
	Y := RST_val;
	state := 0;
ELSIF set THEN
	Y := SET_val;
	state := 0;
ELSIF state > 0 THEN
	(* key has been pushed state machine operating *)
	(* first read the correct input *)
	IF state = 1 THEN
		(* step up *)
		in := su;
	ELSE
		(* step down *)
		in := sd;
	END_IF;
	(* check for single step operation *)
	IF NOT in AND tx - start <= TIME_TO_DWORD(T1) THEN
		Y := Y_start + step;
		state := 0;
	(* check if fast ramp needs to be generated *)
	ELSIF in AND tx - start >= TIME_TO_DWORD(T2) THEN
		Y := Y_start2 + DWORD_TO_REAL(tx - start2) * s2 / speed;
	(* check if slow ramp needs to be generated *)
	ELSIF in AND tx - start >= TIME_TO_DWORD(T1) THEN
		Y := Y_start + DWORD_TO_REAL(tx - start - TIME_TO_DWORD(T1)) * S1 / speed;
		start2 := tx;
		Y_start2 := Y;
	ELSIF NOT in THEN
		state := 0;
	END_IF;
ELSIF su THEN
	(* slow step up *)
	state := 1;
	start := tx;
	step := ss;
	speed := 1000.0;
	Y_start := Y;
ELSIF sd THEN
	(* slow step down *)
	state := 2;
	start := tx;
	step := -ss;
	speed := -1000.0;
	Y_start := Y;
END_IF;

(* make sure output does not exceed limits *)
Y := LIMIT(LIMIT_L, Y, LIMIT_H);

(* revision history
hm	3.11.2007		rev 1.0
	original version

hm	16. mar. 2008	rev 1.1
	added type conversions to avoid warnings under codesys 3.0

hm	11. mar. 2009	rev 1.2
	real constants updated to new systax using dot																																																																																																																																																																																																																																																																																																																																																																																																																																																																																																																																																																																																																																																																																																																																																																																																																																																																																																																																																																																																																																																											

*)

END_FUNCTION_BLOCK

// POUs/Engineering/automation/TUNE2
FUNCTION_BLOCK TUNE2
VAR_INPUT
	SET : BOOL;
	SU, SD : BOOL;
	FU, FD : BOOL;
	RST : BOOL;
END_VAR
VAR_INPUT CONSTANT
	SS : REAL := 0.1;
	FS : REAL := 5.0;
	Limit_L : REAL;
	LIMIT_H : REAL := 100.0;
	RST_val : REAL;
	SET_val : REAL := 100.0;
	TR : TIME := T#500ms;
	S1 : REAL := 2.0;
	S2 : REAL := 10.0;
END_VAR
VAR_OUTPUT
	Y : REAL;
END_VAR
VAR
	tx : DWORD;
	start : DWORD;
	state : INT;
	in : BOOL;
	step : REAL;
	SPEED : REAL;
	Y_start : REAL;
END_VAR

(*
version 1.2	11. mar. 2009
programmer 	hugo
tested by		tobias

tune2 generates an output signal which is set by input switches.
up to 4 switsches can be used to tune the signal up or down.

*)

(* read system time *)
tx := T_PLC_MS();

IF rst THEN
	Y := RST_val;
	state := 0;
ELSIF set THEN
	Y := SET_val;
	state := 0;
ELSIF state > 0 THEN
	(* key has been pushed state machine operating *)
	(* first read the correct input *)
	CASE state OF
		1 :	(* slow up *)
			in := su;
		2 :	(* slow down *)
			in := sd;
		3 :	(* fast up *)
			in := fu;
		4 :	(* fast down *)
			in := fd;
	END_CASE;
	(* check for single step operation *)
	IF NOT in AND tx - start <= TIME_TO_DWORD(TR) THEN
		Y := Y_start + step;
		state := 0;
	(* check if ramp needs to be generated *)
	ELSIF in AND tx - start >= TIME_TO_DWORD(TR) THEN
		Y := Y_start + DWORD_TO_REAL(tx - start - TIME_TO_DWORD(TR)) * speed;
	ELSIF NOT in THEN
		state := 0;
	END_IF;
ELSIF su THEN
	(* slow step up *)
	state := 1;
	start := tx;
	step := ss;
	speed := s1 * 1.0E-3;
	Y_start := Y;
ELSIF sd THEN
	(* slow step down *)
	state := 2;
	start := tx;
	step := -ss;
	speed := -s1 * 1.0E-3;
	Y_start := Y;
ELSIF fu THEN
	(* fast step up *)
	state := 3;
	start := tx;
	step := fs;
	speed := s2 * 1.0E-3;
	y_start := Y;
ELSIF fd THEN
	(* fast step down *)
	state := 4;
	start := tx;
	step := -fs;
	speed := -s2 * 1.0E-3;
	y_start := Y;
END_IF;

(* make sure output does not exceed limits *)
Y := LIMIT(LIMIT_L, Y, LIMIT_H);

(* revision history
hm	3.11.2007		rev 1.0
	original version

hm	16. 3. 2008	rev 1.1
	added type conversions to avoid warnings in codesys 3.0
	improved performance

hm	11. mar. 2009	rev 1.2
	real constants updated to new systax using dot																																																																																																																																																																																																																																																																																																																																																																																																																																																																																																																																																																																																																																																																																																																																																																																																																																																																																																																																																																																																																																																											

*)

END_FUNCTION_BLOCK

// POUs/Mathematical/Vektormathematik/V3_ABS
FUNCTION V3_ABS : REAL
VAR_INPUT
	A : Vector_3;
END_VAR


(*
version 1.0	11 dec 2007
programmer 	hugo
tested by		tobias

this function calculates the length of a vectors in a 3 dimensional space

*)

V3_ABS := SQRT(A.X * A.X + A.Y * A.Y + A.Z * A.Z);


(* revision history
hm		11 dec 2007	rev 1.0
	original version

*)

END_FUNCTION

// POUs/Mathematical/Vektormathematik/V3_ADD
FUNCTION V3_ADD : vector_3
VAR_INPUT
	A : Vector_3;
	B : Vector_3;
END_VAR


(*
version 1.0	11 dec 2007
programmer 	hugo
tested by		tobias

this function adds two vectors in a 3 dimensional space

*)

V3_ADD.X := A.X + B.X;
V3_ADD.Y := A.Y + B.Y;
V3_ADD.Z := A.Z + B.Z;



(* revision history
hm		11 dec 2007	rev 1.0
	original version

*)

END_FUNCTION

// POUs/Mathematical/Vektormathematik/V3_ANG
FUNCTION V3_ANG : REAL
VAR_INPUT
	A : Vector_3;
	B : Vector_3;
END_VAR
VAR
	d : REAL;
END_VAR

(*
version 1.1	10. mar. 2009
programmer 	hugo
tested by		tobias

this function calculates the angle between two vectors in a 3 dimensional space

*)

d := V3_ABS(A) * V3_ABS(B);
IF d > 0 THEN
	V3_ANG := ACOS(LIMIT(-1.0, V3_DPRO(A, B) / d,1.0));
END_IF;

(* revision history
hm	11. dec. 2007	rev 1.0
	original version

hm	10. mar. 2009	rev 1.1
	changed syntax of real constants to 0.0

*)

END_FUNCTION

// POUs/Mathematical/Vektormathematik/V3_DPRO
FUNCTION V3_DPRO : REAL
VAR_INPUT
	A : Vector_3;
	B : Vector_3;
END_VAR


(*
version 1.0	11 dec 2007
programmer 	hugo
tested by		tobias

this function calculates the dot product of two vectors in 3 dimensional space

*)

V3_DPRO := A.X * B.X + A.Y * B.Y + A.Z * B.Z;


(* revision history
hm		11 dec 2007	rev 1.0
	original version

*)

END_FUNCTION

// POUs/Mathematical/Vektormathematik/V3_NORM
FUNCTION V3_NORM : vector_3
VAR_INPUT
	A : Vector_3;
END_VAR
VAR
	la: REAL;
END_VAR

(*
version 1.1	10. mar. 2009
programmer 	hugo
tested by		tobias

this function generates a vectors with absolute length 1 from a vector A in a 3 dimensional space

*)

la := V3_ABS(A);
IF la > 0.0 THEN
	V3_NORM := V3_SMUL(A, 1.0 / la);
END_IF;

(* revision history
hm	11 dec 2007	rev 1.0
	original version

hm	10. mar. 2009	rev 1.1
	changed syntax of real constants to 0.0

*)

END_FUNCTION

// POUs/Mathematical/Vektormathematik/V3_SMUL
FUNCTION V3_SMUL : vector_3
VAR_INPUT
	A : Vector_3;
	M : REAL;
END_VAR


(*
version 1.0	11 dec 2007
programmer 	hugo
tested by		tobias

this function multiplies a vectors in a 3 dimensional space with a skalar M

*)

V3_SMUL.X := A.X * M;
V3_SMUL.Y := A.Y * M;
V3_SMUL.Z := A.Z * M;



(* revision history
hm		11 dec 2007	rev 1.0
	original version

*)

END_FUNCTION

// POUs/Mathematical/Vektormathematik/V3_NUL
FUNCTION V3_NUL : BOOL
VAR_INPUT
	A : Vector_3;
END_VAR


(*
version 1.1	10. mar. 2009
programmer 	hugo
tested by		tobias

this function checks if a vectors in a null Vector

*)

V3_NUL := A.X = 0.0 AND A.Y = 0.0 AND A.Z = 0.0;



(* revision history
hm	12 dec 2007	rev 1.0
	original version

hm	10. mar. 2009	rev 1.1
	changed syntax of real constants to 0.0

*)

END_FUNCTION

// POUs/Mathematical/Vektormathematik/V3_PAR
FUNCTION V3_PAR : BOOL
VAR_INPUT
	A : Vector_3;
	B : Vector_3;
END_VAR


(*
version 1.1	10. mar. 2009
programmer 	hugo
tested by		tobias

this function checks if two vectors in a 3 dimensional space are parallel.
which means the two vectors have the same direction

*)

V3_PAR := V3_ABS(V3_XPRO(A, B)) = 0.0;



(* revision history
hm	11 dec 2007	rev 1.0
	original version

hm	10. mar. 2009	rev 1.1
	changed syntax of real constants to 0.0

*)

END_FUNCTION

// POUs/Mathematical/Vektormathematik/V3_XPRO
FUNCTION V3_XPRO : vector_3
VAR_INPUT
	A : Vector_3;
	B : Vector_3;
END_VAR


(*
version 1.0	11 dec 2007
programmer 	hugo
tested by		tobias

this function adds two vectors in a 3 dimensional space

*)

V3_XPRO.X := A.Y * B.Z - A.Z * B.Y;
V3_XPRO.Y := A.Z * B.X - A.X * B.Z;
V3_XPRO.Z := A.X * B.Y - A.Y * B.X;



(* revision history
hm		11 dec 2007	rev 1.0
	original version

*)

END_FUNCTION

// POUs/Mathematical/Vektormathematik/V3_REV
FUNCTION V3_REV : vector_3
VAR_INPUT
	A : Vector_3;
END_VAR


(*
version 1.0	11 dec 2007
programmer 	hugo
tested by		tobias

this function reverses a vector in a 3 dimensional space

*)

V3_REV.X := -A.X;
V3_REV.Y := -A.Y;
V3_REV.Z := -A.Z;



(* revision history
hm		11 dec 2007	rev 1.0
	original version

*)

END_FUNCTION

// POUs/Mathematical/Vektormathematik/V3_SUB
FUNCTION V3_SUB : vector_3
VAR_INPUT
	A : Vector_3;
	B : Vector_3;
END_VAR


(*
version 1.0	11 dec 2007
programmer 	hugo
tested by		tobias

this function subtracts two vectors in a 3 dimensional space
V3_SUB = A - B

*)

V3_SUB.X := A.X - B.X;
V3_SUB.Y := A.Y - B.Y;
V3_SUB.Z := A.Z - B.Z;



(* revision history
hm		11 dec 2007	rev 1.0
	original version

*)

END_FUNCTION

// POUs/Mathematical/Vektormathematik/V3_XANG
FUNCTION V3_XANG : REAL
VAR_INPUT
	A : Vector_3;
END_VAR
VAR
	la: REAL;
END_VAR

(*
version 1.1	10. mar. 2009
programmer 	hugo
tested by		tobias

this function calculates the angle between the X-axis and a vectors in a 3 dimensional space

*)

la := V3_ABS(a);
IF la > 0.0 THEN
	V3_XANG := ACOS(A.X / la);
END_IF;

(* revision history
hm	11 dec 2007	rev 1.0
	original version

hm	10. mar. 2009	rev 1.1
	changed syntax of real constants to 0.0

*)

END_FUNCTION

// POUs/Mathematical/Vektormathematik/V3_YANG
FUNCTION V3_YANG : REAL
VAR_INPUT
	A : Vector_3;
END_VAR
VAR
	la: REAL;
END_VAR

(*
version 1.1	10. mar. 2009
programmer 	hugo
tested by		tobias

this function calculates the angle between the Y-axis and a vectors in a 3 dimensional space

*)

la := V3_ABS(a);
IF la > 0.0 THEN
	V3_YANG := ACOS(A.Y / la);
END_IF;

(* revision history
hm	11 dec 2007	rev 1.0
	original version

hm	10. mar. 2009	rev 1.1
	changed syntax of real constants to 0.0

*)

END_FUNCTION

// POUs/Mathematical/Vektormathematik/V3_ZANG
FUNCTION V3_ZANG : REAL
VAR_INPUT
	A : Vector_3;
END_VAR
VAR
	la: REAL;
END_VAR

(*
version 1.1	10. mar. 2009
programmer 	hugo
tested by		tobias

this function calculates the angle between the Z-axis and a vectors in a 3 dimensional space

*)

la := V3_ABS(a);
IF la > 0.0 THEN
	V3_ZANG := ACOS(A.Z / la);
END_IF;

(* revision history
hm	11 dec 2007	rev 1.0
	original version

hm	10. mar. 2009	rev 1.1
	changed syntax of real constants to 0.0

*)

END_FUNCTION

// POUs/Building/HLK/WATER_CP
FUNCTION WATER_CP : REAL
VAR_INPUT
	T : REAL;
END_VAR
VAR
	Pts : INT := 10;
	data : ARRAY[1..20, 0..1] OF REAL :=[ 0.0,4.228, 5.0,4.20, 10.0,4.188, 15.0,4.184, 50.0,4.181, 60.0,4.183, 70.0,4.187, 80.0,4.194, 90.0,4.204, 100.0,4.22];
END_VAR

(*
version 1.2	13. mar. 2009
programmer 	hugo
tested by		tobias

water_cp calculates the specific heat capacity of liquid water from 0..100 °C 

*)

WATER_CP := LINEAR_INT(T, Data, Pts);


(*
    °C - die Celsius-Temperatur in Grad Celsius
    v  das spezifische Volumen in Kubikdezimeter je Kilogramm dm³/kg
    h  die spezifische Enthalpie in Kilojoule je Kilogramm 	kJ/kg
    u  die spezifische Innere Energie in Kilojoule je Kilogramm 	kJ/kg
    s  die spezifische Entropie in Kilojoule je Kilogramm mal Kelvin 	kJ/(kg·K)
    cp - die spezifische Wärmekapazität bei konstantem Druck in Kilojoule je Kilogramm mal Kelvin 	kJ/(kg·K)
    Y  Volumenausdehnungskoeffizient in 10-3 durch Kelvin  10-3/K
    L  Wärmeleitfähigkeit in Milliwatt je Meter mal Kelvin  mW / (m·K) 
    n  Viskosität in Mikropascal mal Sekunde uPa·s 	
    s ?  Oberflächenspannung in Millinewton je Meter  mN/m


°C 		v 				h 			u 		s 			cp 		Y 		L		n		s	
-20		1,006580	
0 		1,000160 		0,06 		-0,04 	-0,0001 	4,228 	-0,080 	561,0 	1792 	75,65
4		1,000028
5 		1,0000 		21,1 		21,0 	0,076 		4,200 	0,011 	570,6 	1518 	74,95
10 		1,0003 		42,1 		42,0 	0,151 		4,188 	0,087 	580,0 	1306 	74,22
15 		1,0009 		63,0 		62,9 	0,224 		4,184 	0,152 	589,4 	1137 	73,49
20 		1,001797 		83,9 		83,8 	0,296 		4,183 	0,209 	598,4 	1001 	72,74
25 		1,0029 		104,8 		104,7 	0,367 		4,183 	0,259 	607,2 	890,4 	71,98
30 		1,0044 		125,8 		125,7 	0,437 		4,183 	0,305 	615,5 	797,7 	71,20
35 		1,0060 		146,7 		146,6 	0,505 		4,183 	0,347 	623,3 	719,6 	70,41
40 		1,007842 		167,58 	167,5 	0,572 		4,182 	0,386 	630,6 	653,3 	69,60
45 		1,0099 		188,5 		188,4 	0,638 		4,182 	0,423 	637,3 	596,3 	68,78
50 		1,0121 		209,4 		209,3 	0,704 		4,181 	0,457 	643,6 	547,1 	67,95
60 		1,017089 		251,2 		251,1 	0,831 		4,183 	0,522 	654,4 	466,6 	66,24
70 		1,0227 		293,1 		293,0 	0,955 		4,187 	0,583 	663,1 	404,1 	64,49
80 		1,029027 		335,0 		334,9 	1,075 		4,194 	0,640 	670,0 	354,5 	62,68
90 		1,0359 		377,0 		376,9 	1,193 		4,204 	0,696 	675,3 	314,6 	60,82
99,63 	1,0431 		417,5 		417,4 	1,303 		4,217 	0,748 	679,0 	283,0 	58,99
100	1,043453		419,1

Stoffdaten von Wasser Quelle Wickipedia

Wasser hat unter Normaldruck seine größte Dichte von 1000 Kilogramm pro Kubikmeter bei 3,98 °C und zeigt damit eine Dichteanomalie. 
Diese besteht darin, dass sich Wasser unterhalb von 3,98 °C bei weiterer Temperaturverringerung, auch beim Wechsel zum festen 
Aggregatzustand, wieder ausdehnt, was man nur von wenigen Stoffen kennt. Die derzeit genauesten publizierten Werte für die maximale 
Dichte liegen bei (999,974950 ± 0,00084) kg/m³ und bei (3,983 ± 0,00067) °C für die Temperatur, bei der dieser Wert erreicht wird. 
Die Werte stellen einen Mittelwert der von verschiedenen physikalischen Instituten veröffentlichten Zahlen dar (Stand 2001).

Die Berechnung der Dichte von luftfreiem Wasser DLF in Abhängigkeit von der Temperatur T ([T] = °C) kann mit Hilfe der folgenden 
Virialgleichung erfolgen:
: \frac{D_{\rm LF}}{\rm g/l} = \frac{a_0 + a_1 T + a_2 T^2 + a_3 T^3 + a_4 T^4 + a_5 T^5}{1 + b T}.
mit den Koeffizienten: a0 = 999,83952; a1 = 16,952577 (°C)-1; a2 = -7,9905127·10-3 (°C)-2; a3 = -4,6241757·10-5 (°C)-3; 
a4 = 1,0584601·10-7 (°C)-4; a5 = -2,8103006·10-10 (°C)-5 und b = 0,0168872. 
Für die Berechnung der Dichte von luftgesättigtem Wasser korrigiert man den Wert nach 
DLG/(g/l) = DLF/(g/l) - 0,004612 + 0,000106 (°C)-1·T. (Quelle: PTB-Mitteilungen 100/3-90)

*)

(* revision history

hm	29.10.2007	rev 1.0
	original version

hm	27. dec 2007	rev 1.1
	increased accuracy

hm	13. mar. 2009	rev 1.2
	real constants updated to new systax using dot

*)

END_FUNCTION

// POUs/Building/HLK/WCT
FUNCTION WCT : REAL
VAR_INPUT
	T : REAL;
	V : REAL;
END_VAR


(*
version 1.2	13. mar. 2009
programmer 	hugo
tested by		tobias

this function calculates the wind chill temperature

*)

IF V < 5.0 OR T > 10.0 THEN
	WCT := T;
ELSE
	WCT := 13.12 + 0.6215 * T +(0.3965 * T - 11.37) * EXP(LN(v) * 0.16);
END_IF;


(* revision history
hm	7 feb 2007		rev 1.0
	original version

hm	7 dec 2007	rev 1.1
	changed code for better performance

hm	13. mar. 2009	rev 1.2
	real constants updated to new systax using dot

*)

END_FUNCTION

// POUs/Mathematical/WINDOW2
FUNCTION WINDOW2 : BOOL
VAR_INPUT
	low : REAL;
	in : REAL;
	high : REAL;
END_VAR


(*
	version 1.0	31 oct 2007
	programmer 	hugo
	tested BY	tobias

this checks a signal if the signal is between the upper and lower limit including the two limits
*)

WINDOW2 := in <= high AND in >= low;


(* revision history
hm	31.10.2007	rev 1.0
	original version

*)

END_FUNCTION

// POUs/Logic/gate logic/WORD_OF_BYTE
FUNCTION WORD_OF_BYTE : WORD
VAR_INPUT
	B1 : BYTE;
	B0 : BYTE;
END_VAR


(*
version 1.4	18. jul. 2009
programmer 	hugo
tested by		tobias

this function creates a word from 2 individual bytes

*)

WORD_OF_BYTE := SHL(BYTE_TO_WORD(B1),8) OR BYTE_TO_WORD(B0);

(* revision history
hm	24. jan 2007	rev 1.0
	original version

hm	2. jan 2008	rev 1.1
	improved performance

hm	19. feb 2008	rev 1.2
	replaced and with or for better compatibility

hm	23. apr. 2008	rev 1.3
	reverse order of inputs to be more logical

hm	18. jul. 2009	rev 1.4
	added type conversions for compatibility reasons

*)

END_FUNCTION

// POUs/Logic/gate logic/WORD_OF_DWORD
FUNCTION WORD_OF_DWORD : WORD
VAR_INPUT
	in : DWORD;
	N : BYTE;
END_VAR


(*
version 1.2	30. oct. 2008
programmer 	hugo
tested by	oscat

this function extracts a single word from the nth position from right (right is lowest byte)
the lower word (starting with Bit0 from in) is selected with N=0.
*)

WORD_OF_DWORD := DWORD_TO_WORD(SHR(in,SHL(n,4)));

(* revision history
hm	17. jan 2007	rev 1.0
	original version

hm	2. jan 2008		rev 1.1
	improved performance

hm	30. oct. 2008	rev 1.2
	improved performance
*)

END_FUNCTION

// POUs/Engineering/signal processing/WORD_TO_RANGE
FUNCTION WORD_TO_RANGE : REAL
VAR_INPUT
	X : WORD;
	low : REAL;
	high : REAL;
END_VAR


(*
version 1.1	10. mar. 2009
programmer 	hugo
tested by		tobias

Word_to_Range converts a Byte into a real between low and high.

*)

WORD_TO_RANGE := (high - low) * WORD_TO_REAL(X) * 0.00001525902189669640 + low;


(* revision history
hm	9. jan 2008	rev 1.0
	original version

hm	10. mar. 2009	rev 1.1
	improved code
*)

END_FUNCTION
